FUNCTION_BLOCK Feeder (* Basic Function Block Type *)
  (* Standard: 61499-2 *)
  (* Version 0.0, 1/9/2024, Cheyan, Schneider Electric, Template *)
  PACKAGE Main;
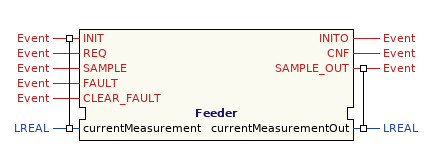
  EVENT_INPUT
    INIT WITH currentMeasurement;
    REQ;
    SAMPLE;
    FAULT;
    CLEAR_FAULT;
  END_EVENT
  EVENT_OUTPUT
    INITO; (* Initialization Confirm *)
    CNF; (* Execution Confirmation *)
    SAMPLE_OUT WITH currentMeasurementOut;
  END_EVENT
  VAR_INPUT
    currentMeasurement : LREAL; (* Input event qualifier *)
  END_VAR
  VAR_OUTPUT
    currentMeasurementOut : LREAL; (* Output event qualifier *)
  END_VAR
  VAR
    currentInternal : LREAL;
  END_VAR
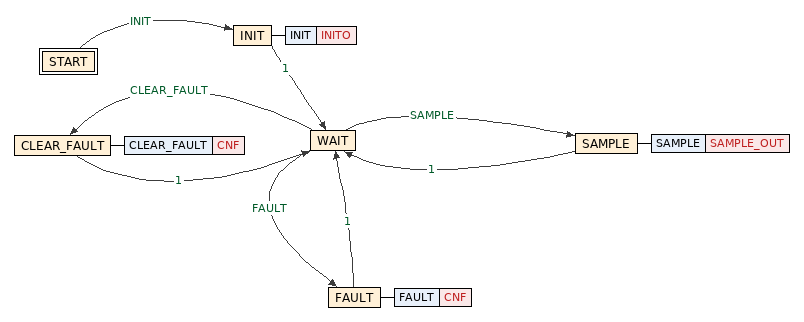
  EC_STATES
    START; (* Initial State *)
    INIT : INIT -> INITO; (* Initialization *)
    WAIT;
    SAMPLE : SAMPLE -> SAMPLE_OUT;
    FAULT : FAULT -> CNF;
    CLEAR_FAULT : CLEAR_FAULT -> CNF;
  END_STATES
  EC_TRANSITIONS
    INIT TO WAIT := 1;
    WAIT TO SAMPLE := SAMPLE;
    SAMPLE TO WAIT := 1;
    WAIT TO FAULT := FAULT;
    FAULT TO WAIT := 1;
    WAIT TO CLEAR_FAULT := CLEAR_FAULT;
    CLEAR_FAULT TO WAIT := 1;
    START TO INIT := INIT;
  END_TRANSITIONS
  ALGORITHM INIT IN ST: (* Initialization algorithm Setting the initial current measurement of the Feeder *)
;

currentInternal := currentMeasurement;
  END_ALGORITHM
  ALGORITHM REQ IN ST: (* Normally executed algorithm *)
;
  END_ALGORITHM
  ALGORITHM SAMPLE IN ST: (* Sending out current measurement *)
;

currentMeasurementOut := currentInternal;
  END_ALGORITHM
  ALGORITHM FAULT IN ST: (* Triggering fault current. Fault current set at 1.5x of the normal current *)
;

currentInternal := currentMeasurement + currentMeasurement/2;
  END_ALGORITHM
  ALGORITHM CLEAR_FAULT IN ST:
;

currentInternal := 0;
  END_ALGORITHM
END_FUNCTION_BLOCK
